
FUNCTION CB_abs_dint : DINT


TITLE = ' Absolute value of a number '
VERSION : '1.0'
AUTHOR  : CB
NAME    : abs_dint
FAMILY  : TNI

VAR_INPUT
    IN : DINT;
END_VAR

VAR_TEMP

END_VAR

BEGIN

CB_abs_dint := ABS(IN);

END_FUNCTION
